FUNCTION_BLOCK SystemData
VAR_INPUT
	netID: T_AmsNetID;
END_VAR
VAR_OUTPUT
	TimeIsRunning: BOOL;
	
	MachineTime: DT;
	MachineSystemTime: TIMESTRUCT;
END_VAR
VAR
	GetTime: NT_GetTime;
	synchTime: TON;
	
	F_Trig_RTC: F_Trig;
	DataRTC: RTC;
END_VAR

VAR CONSTANT
	TimerCheck: TIME := T#2s;
END_VAR

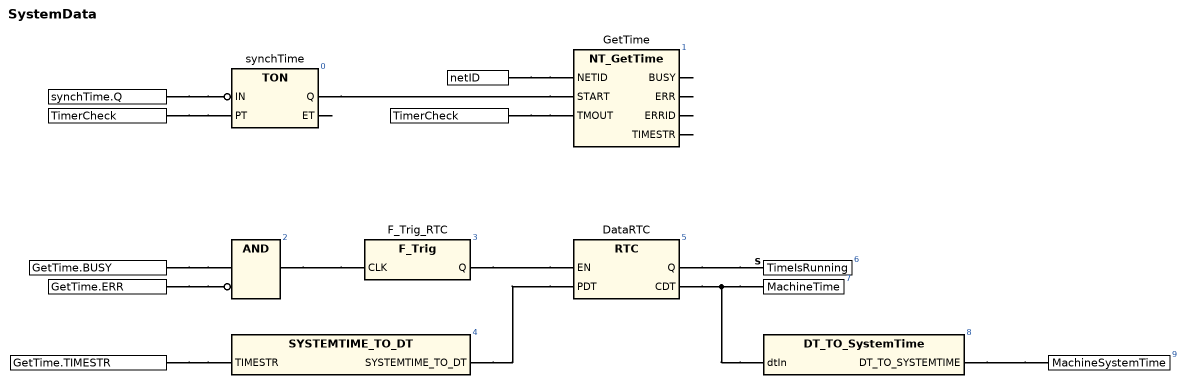
synchTime(IN := NOT synchTime.Q, PT := TimerCheck); // TON
GetTime(NETID := netID, START := synchTime.Q, TMOUT := TimerCheck); // NT_GetTime
F_Trig_RTC(CLK := GetTime.BUSY AND NOT GetTime.ERR); // F_Trig
DataRTC(EN := F_Trig_RTC.Q, PDT := SYSTEMTIME_TO_DT(TIMESTR := GetTime.TIMESTR)); // RTC
TimeIsRunning S= DataRTC.Q;
MachineTime := DataRTC.CDT;
MachineSystemTime := DT_TO_SystemTime(dtIn := DataRTC.CDT);

END_FUNCTION_BLOCK

(* stored: Version 1.1.0.1, ProductVersion 3.1.4024.6
   POU SystemData: Id {90f20abf-b74f-44a4-a448-7d4c17aa528d}, SpecialFunc None *)
